// TIA Portal V17 export
BLOCK "CompleteRestart"   // ObjectSW100, LAD
BEGIN
END_BLOCK
